{attribute 'qualified_only'}

TYPE eInputSignal :
(
	None 			:= 	0,
	GenLowFuel 		:= 	1,
	StopOperation 	:= 	2,
	EMstop			:=	3
) UINT;
END_TYPE

(* stored: Version 1.1.0.1, ProductVersion 3.1.4026.18
   DUT eInputSignal: Id {426d2b47-903a-4004-91ab-ee8d00ebd04e} *)
